INTERFACE I_UndulatorComplex

PROPERTY rCurrentPhotonEnergy : LREAL
GET
END_GET
END_PROPERTY

PROPERTY rTargetPhotonEnergy : LREAL
GET
END_GET
END_PROPERTY

END_INTERFACE

(* stored: Version 1.1.0.1, ProductVersion 3.1.4026.11
   Itf I_UndulatorComplex: Id {58c10c85-f752-4da9-8bb8-c4aa0534b71a}
   Property rCurrentPhotonEnergy: Id {13076688-de6c-46fb-bc96-f35dd9b5072c}
   Get Get: Id {7e3c5a1a-1015-44fc-886d-8c84bff5e2e7}
   Property rTargetPhotonEnergy: Id {3d22f590-84aa-487e-934d-179d4b5d185d}
   Get Get: Id {3960bfc6-ae2c-4d6a-8d87-eb5698cebc8f} *)
